{attribute 'qualified_only'}
{attribute 'strict'}
TYPE ENUM_OrderState :
(
	Working := 0,
	Done	:= 1
);
END_TYPE

(* stored: Version 1.1.0.1, ProductVersion 3.1.4024.9
   DUT ENUM_OrderState: Id {279fda47-cecd-4877-9fee-6b34a5ec57c2} *)
